FUNCTION_BLOCK container_two_basic
  (* Standard: 61499-2 *)
  (* Version 0.1, 2017-00-14, Hammond, HAMMONDSDESKTOP *)
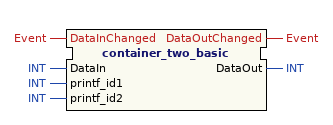
  EVENT_INPUT
    DataInChanged;
  END_EVENT
  EVENT_OUTPUT
    DataOutChanged;
  END_EVENT
  VAR_INPUT
    DataIn : INT;
    printf_id1 : INT;
    printf_id2 : INT;
  END_VAR
  VAR_OUTPUT
    DataOut : INT;
  END_VAR
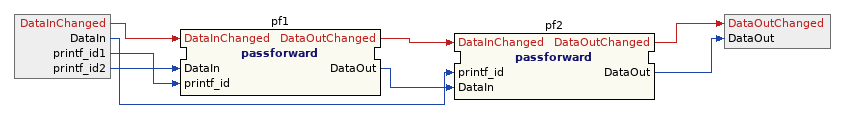
  FBS
    pf1 : passforward;
    pf2 : passforward;
  END_FBS
  EVENT_CONNECTIONS
    DataInChanged TO pf1.DataInChanged;
    pf2.DataOutChanged TO DataOutChanged;
    pf1.DataOutChanged TO pf2.DataInChanged;
  END_CONNECTIONS
  DATA_CONNECTIONS
    DataIn TO pf1.DataIn;
    printf_id1 TO pf1.printf_id;
    printf_id2 TO pf2.printf_id;
    pf2.DataOut TO DataOut;
    pf1.DataOut TO pf2.DataIn;
  END_CONNECTIONS
END_FUNCTION_BLOCK
